VAR_GLOBAL CONSTANT
	PLCPRJ_BUFFER_SIZE					: UDINT := 1000;(* Max. internal fifo/receiver buffer size *)

	(* Some project specific error codes *)
	PLCPRJ_ERROR_SENDFIFO_OVERFLOW		: UDINT := 16#8103;
	PLCPRJ_ERROR_RECFIFO_OVERFLOW		: UDINT := 16#8104;
END_VAR

(* stored: Version 1.1.0.1, ProductVersion 3.1.0.20
   GVL Global_Variables: Id {0cdf50cb-6348-4d09-8f82-3be1b63416b2} *)
